ABB RAPID module: 002450D5

MODULE Module1
    CONST robtarget PickUp:=[[114.467979448,162.108018639,169.267197731],[0.400706229,-0.400706048,-0.58261,-0.582610305],[-1,-2,2,1],[9E+09,9E+09,9E+09,9E+09,9E+09,9E+09]];
    CONST robtarget DropOff:=[[114.529328973,955.01069365,260.246517958],[0.40070622,-0.400705989,-0.582609862,-0.58261049],[0,-1,1,0],[9E+09,9E+09,9E+09,9E+09,9E+09,9E+09]];
ENDMODULE
